FUNCTION_BLOCK PhaseBasic (* Basic Function Block Type *)
  (* Standard: 61499-2 *)
  (* Version 0.0, 6/4/2026, Schneider Electric, Template *)
  PACKAGE SE.Nereda;
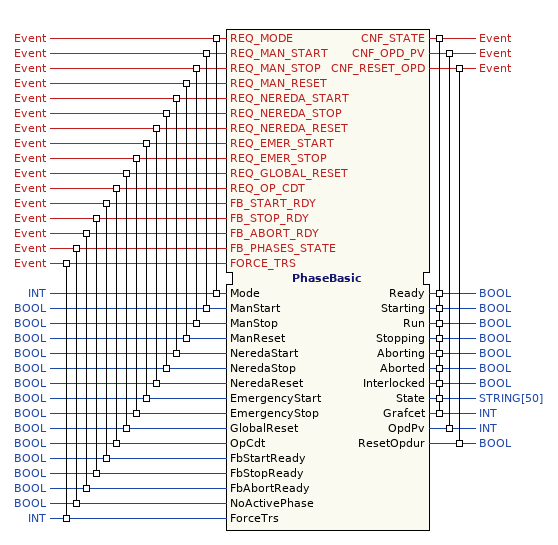
  EVENT_INPUT
    REQ_MODE WITH Mode;
    REQ_MAN_START WITH ManStart;
    REQ_MAN_STOP WITH ManStop;
    REQ_MAN_RESET WITH ManReset;
    REQ_NEREDA_START WITH NeredaStart;
    REQ_NEREDA_STOP WITH NeredaStop;
    REQ_NEREDA_RESET WITH NeredaReset;
    REQ_EMER_START WITH EmergencyStart;
    REQ_EMER_STOP WITH EmergencyStop;
    REQ_GLOBAL_RESET WITH GlobalReset;
    REQ_OP_CDT WITH OpCdt;
    FB_START_RDY WITH FbStartReady;
    FB_STOP_RDY WITH FbStopReady;
    FB_ABORT_RDY WITH FbAbortReady;
    FB_PHASES_STATE WITH NoActivePhase;
    FORCE_TRS WITH ForceTrs;
  END_EVENT
  EVENT_OUTPUT
    CNF_STATE WITH Interlocked, Ready, Starting, Run, Stopping, Aborting, Aborted, State, Grafcet;
    CNF_OPD_PV WITH OpdPv;
    CNF_RESET_OPD WITH ResetOpdur;
  END_EVENT
  VAR_INPUT
    Mode : INT;
    ManStart : BOOL;
    ManStop : BOOL;
    ManReset : BOOL;
    NeredaStart : BOOL;
    NeredaStop : BOOL;
    NeredaReset : BOOL;
    EmergencyStart : BOOL;
    EmergencyStop : BOOL;
    GlobalReset : BOOL;
    OpCdt : BOOL;
    FbStartReady : BOOL;
    FbStopReady : BOOL;
    FbAbortReady : BOOL;
    NoActivePhase : BOOL;
    ForceTrs : INT;
  END_VAR
  VAR_OUTPUT
    Ready : BOOL;
    Starting : BOOL;
    Run : BOOL;
    Stopping : BOOL;
    Aborting : BOOL;
    Aborted : BOOL;
    Interlocked : BOOL;
    State : STRING[50];
    Grafcet : INT;
    OpdPv : INT;
    ResetOpdur : BOOL;
  END_VAR
  VAR
    MemoMode : INT;
  END_VAR
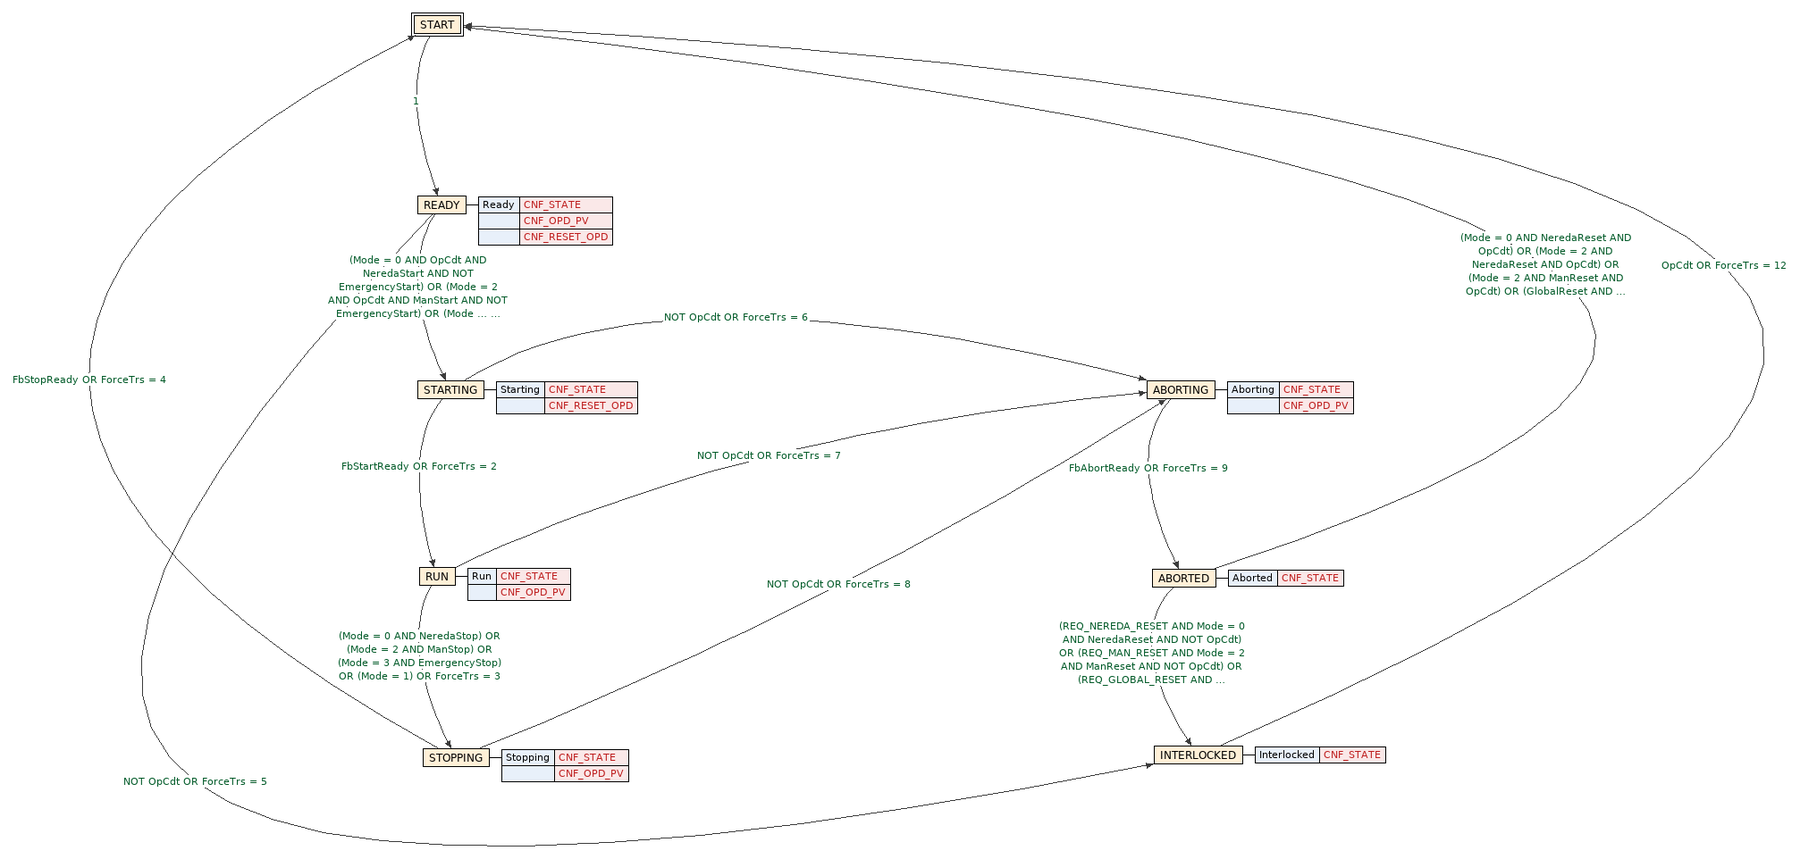
  EC_STATES
    START; (* Initial State *)
    READY : Ready -> CNF_STATE, -> CNF_OPD_PV, -> CNF_RESET_OPD;
    STARTING : Starting -> CNF_STATE, -> CNF_RESET_OPD;
    RUN : Run -> CNF_STATE, -> CNF_OPD_PV;
    STOPPING : Stopping -> CNF_STATE, -> CNF_OPD_PV;
    ABORTING : Aborting -> CNF_STATE, -> CNF_OPD_PV;
    ABORTED : Aborted -> CNF_STATE;
    INTERLOCKED : Interlocked -> CNF_STATE;
  END_STATES
  EC_TRANSITIONS
    READY TO INTERLOCKED := NOT OpCdt OR ForceTrs = 5;
    STARTING TO ABORTING := NOT OpCdt OR ForceTrs = 6;
    RUN TO ABORTING := NOT OpCdt OR ForceTrs = 7;
    STOPPING TO ABORTING := NOT OpCdt OR ForceTrs = 8;
    INTERLOCKED TO START := OpCdt OR ForceTrs = 12;
    START TO READY := 1;
    READY TO STARTING := (Mode = 0 AND OpCdt AND NeredaStart AND NOT EmergencyStart) OR (Mode = 2 AND OpCdt AND ManStart AND NOT EmergencyStart) OR (Mode = 3 AND OpCdt AND EmergencyStart AND NoActivePhase) OR ForceTrs = 1;
    STARTING TO RUN := FbStartReady OR ForceTrs = 2;
    RUN TO STOPPING := (Mode = 0 AND NeredaStop) OR (Mode = 2 AND ManStop) OR (Mode = 3 AND EmergencyStop) OR (Mode = 1) OR ForceTrs = 3;
    ABORTING TO ABORTED := FbAbortReady OR ForceTrs = 9;
    ABORTED TO INTERLOCKED := (REQ_NEREDA_RESET AND Mode = 0 AND NeredaReset AND NOT OpCdt) OR (REQ_MAN_RESET AND Mode = 2 AND ManReset AND NOT OpCdt) OR (REQ_GLOBAL_RESET AND GlobalReset AND NOT OpCdt) OR ForceTrs = 11;
    STOPPING TO START := FbStopReady OR ForceTrs = 4;
    ABORTED TO START := (Mode = 0 AND NeredaReset AND OpCdt) OR (Mode = 2 AND NeredaReset AND OpCdt) OR (Mode = 2 AND ManReset AND OpCdt) OR (GlobalReset AND OpCdt) OR ForceTrs = 10;
  END_TRANSITIONS
  ALGORITHM Starting IN ST:
;
MemoMode := Mode;

Ready := FALSE;
Starting := TRUE;
Run := FALSE;
Stopping := FALSE;
Aborting := FALSE;
Aborted := FALSE;
Interlocked := FALSE;
State := 'Starting';
Grafcet := 1;
ResetOpdur := FALSE;
  END_ALGORITHM
  ALGORITHM Ready IN ST:
;
Ready := TRUE;
Starting := FALSE;
Run := FALSE;
Stopping := FALSE;
Aborting := FALSE;
Aborted := FALSE;
Interlocked := FALSE;
State := 'Ready';
Grafcet := 0;
OpdPv := 0;
ResetOpdur := TRUE;
  END_ALGORITHM
  ALGORITHM Run IN ST:
;
Ready := FALSE;
Starting := FALSE;
Run := TRUE;
Stopping := FALSE;
Aborting := FALSE;
Aborted := FALSE;
Interlocked := FALSE;
State := 'Running';
Grafcet := 2;
OpdPv := 1;
  END_ALGORITHM
  ALGORITHM Stopping IN ST:
;
Ready := FALSE;
Starting := FALSE;
Run := FALSE;
Stopping := TRUE;
Aborting := FALSE;
Aborted := FALSE;
Interlocked := FALSE;
State := 'Stopping';
Grafcet := 3;
OpdPv := 0;
  END_ALGORITHM
  ALGORITHM Aborting IN ST:
;
Ready := FALSE;
Starting := FALSE;
Run := FALSE;
Stopping := FALSE;
Aborting := TRUE;
Aborted := FALSE;
Interlocked := FALSE;
State := 'Aborting';
Grafcet := 5;
OpdPv := 0;
  END_ALGORITHM
  ALGORITHM Aborted IN ST:
;
Ready := FALSE;
Starting := FALSE;
Run := FALSE;
Stopping := FALSE;
Aborting := FALSE;
Aborted := TRUE;
Interlocked := FALSE;
State := 'Aborted';
Grafcet := 6;
  END_ALGORITHM
  ALGORITHM Interlocked IN ST:
;
Ready := FALSE;
Starting := FALSE;
Run := FALSE;
Stopping := FALSE;
Aborting := FALSE;
Aborted := FALSE;
Interlocked := TRUE;
State := 'Interlocked';
Grafcet := 7;
  END_ALGORITHM
END_FUNCTION_BLOCK
